INTERFACE I_JsonDeserializerDisposedEvent EXTENDS I_Event

PROPERTY PUBLIC Target : I_JsonDeserializer
GET
END_GET
END_PROPERTY

END_INTERFACE

(* stored: Version 1.1.0.1, ProductVersion 3.1.4024.12
   Itf I_JsonDeserializerDisposedEvent: Id {3318f30e-cc8f-48da-815c-aa22cd75b2a9}
   Property Target: Id {b0f28433-6ee6-4ae3-b89d-b21754f0443c}
   Get Get: Id {d141094d-0fe7-487c-9179-4ac505f8fe09} *)
